FUNCTION_BLOCK MC_AxisControl
VAR_INPUT	
END_VAR
VAR_IN_OUT
	axisRef			: AXIS_REF;
END_VAR
VAR_OUTPUT
END_VAR
VAR
	// Controls
	bEnable				: BOOL;
	bReset				: BOOL;
	bMove				: BOOL;
	                	
	// Statuses     	
	bEnabled			: BOOL;
	bReferenced			: BOOL;
	bError				: BOOL;
	nErrorID			: UDINT;
	bMoveDone			: BOOL;
	bInPosition			: BOOL;
	nActualPosition		: LREAL;
	nActualVelocity		: LREAL;
	
	// Settings
	nTargetPosition		: LREAL;
	nTargetVelocity		: LREAL;
	nTargetAcceleration	: LREAL;
	
	fbEnable			: MC_Power;
	fbMove				: MC_MoveAbsolute;
	fbReset				: MC_Reset;
	fbActualPosition	: MC_ReadActualPosition;
	fbActualVelocity	: MC_ReadActualVelocity;
	
	trigErrorSet		: R_TRIG;
	trigErrorReSet		: R_TRIG;
	trigMoveDone		: R_TRIG;
END_VAR

// Power On
fbEnable(
	Axis:= axisRef, 
	Enable:= bEnable, 
	Enable_Positive:= bEnable, 
	Enable_Negative:= bEnable, 
	Override:= , 
	BufferMode:= , 
	Options:= , 
	Status=> bEnabled, 
	Busy=> , 
	Active=> , 
	Error=> , 
	ErrorID=> );
	
// Reset
fbReset(
	Axis:= axisRef, 
	Execute:= bReset, 
	Done=> , 
	Busy=> , 
	Error=> , 
	ErrorID=> );
	
// Move Absolute
fbMove(
	Axis:= axisRef, 
	Execute:= bMove AND bEnabled, 
	Position:= nTargetPosition, 
	Velocity:= nTargetVelocity, 
	Acceleration:= nTargetAcceleration, 
	Deceleration:= nTargetAcceleration, 
	Jerk:= , 
	BufferMode:= , 
	Options:= , 
	Done=> bMoveDone, 
	Busy=> , 
	Active=> , 
	CommandAborted=> , 
	Error=> , 
	ErrorID=> );
	
// Status Actual Position
fbActualPosition(
	Axis:= axisRef, 
	Enable:= TRUE, 
	Valid=> , 
	Busy=> , 
	Error=> , 
	ErrorID=> , 
	Position=> nActualPosition);

// Status Actual Velocity	
fbActualVelocity(
	Axis:= axisRef, 
	Enable:= TRUE, 
	Valid=> , 
	Busy=> , 
	Error=> , 
	ErrorID=> , 
	ActualVelocity=> nActualVelocity);
	
// In Position	
trigMoveDone(CLK := bMoveDone);
IF trigMoveDone.Q 
AND ABS(nTargetPosition - nActualPosition) < 0.1 
THEN
	bMove := FALSE;
	bInPosition := TRUE;
ELSIF ABS(nTargetPosition - nActualPosition) > 0.1 THEN
	bInPosition := FALSE;
END_IF

// Error Detection
trigErrorSet(CLK:= fbEnable.Error OR fbReset.Error OR fbMove.Error OR fbActualPosition.Error OR fbActualVelocity.Error, Q=> );
trigErrorReSet(CLK:= NOT fbEnable.Error AND NOT fbReset.Error AND NOT fbMove.Error AND NOT fbActualPosition.Error AND NOT fbActualVelocity.Error, Q=> );
IF trigErrorSet.Q THEN
	bError := TRUE;
	bEnable := FALSE;
	nErrorID := fbEnable.ErrorID + fbReset.ErrorID + fbMove.ErrorID + fbActualPosition.ErrorID + fbActualVelocity.ErrorID;
END_IF
IF trigErrorReSet.Q THEN
	bError := FALSE;
	bReset := FALSE;
	nErrorID := 0;
END_IF

END_FUNCTION_BLOCK

(* stored: Version 1.1.0.1, ProductVersion 3.1.4024.9
   POU MC_AxisControl: Id {84cc6ef7-9ee1-4c68-b55b-f1fda5149a92}, SpecialFunc None *)
